Yaskawa INFORM job: TWIN_FRONT_WELD_90ST-2_5340.JBI

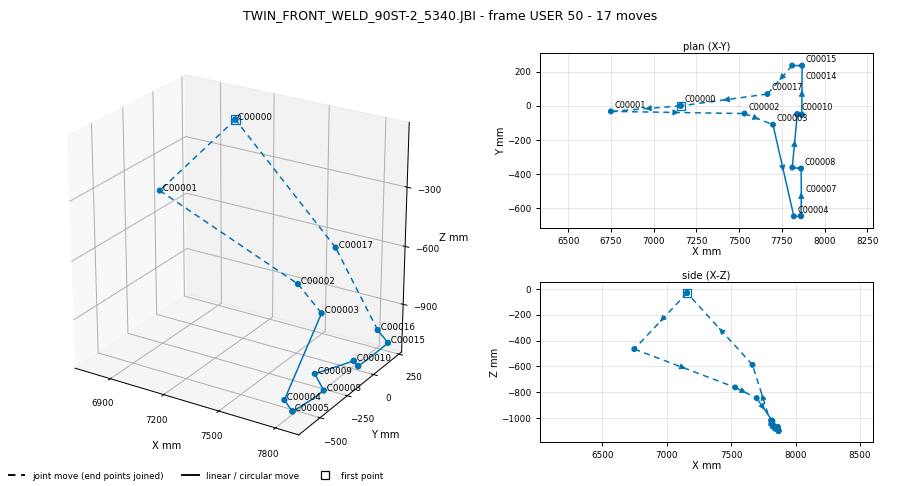
[picture p0: tool path of TWIN_FRONT_WELD_90ST-2_5340.JBI in frame USER 50, 17 of 19 moves have a stored position in this frame; points joined in program order, loops and branches not executed]
/JOB
//NAME TWIN_FRONT_WELD_90ST-2_5340
///FOLDERNAME 02-SKRZYNIE_JOBS
//POS
///NPOS 19,19,0,4,0,0
///USER 50
///TOOL 0
///POSTYPE USER
///RECTAN
///RCONF 0,0,1,0,0,0,0,0,0,0,0,0,0,0,0,0,0,0,0,0,0,0,0,0
C00000=7158.107,0.308,-30.113,-0.0036,-53.6521,0.0034
///RCONF 1,0,1,0,0,0,0,0,0,0,0,0,0,0,0,0,0,0,0,0,0,0,0,0
C00001=6749.261,-32.286,-465.417,15.1595,35.6819,-145.6807
///RCONF 1,0,0,0,0,0,0,0,0,0,0,0,0,0,0,0,0,0,0,0,0,0,0,0
C00002=7531.538,-44.927,-762.719,8.7291,34.6461,-164.2133
C00003=7698.169,-109.933,-845.445,15.9625,40.0165,-157.0814
///RCONF 0,0,0,0,0,0,0,0,0,0,0,0,0,0,0,0,0,0,0,0,0,0,0,0
C00004=7820.412,-646.733,-1023.988,41.9712,23.9862,-139.0909
C00005=7861.855,-645.939,-1070.027,41.9679,23.9849,-139.0942
C00006=7861.883,-644.400,-1070.166,41.9241,23.9457,-138.9976
C00007=7863.853,-523.749,-1081.452,38.5881,21.3794,-131.1067
C00008=7862.327,-366.605,-1089.610,38.1696,21.1192,-130.0311
C00009=7811.247,-360.951,-1020.499,38.1489,21.1058,-129.9915
C00010=7840.461,-48.547,-1081.078,15.4598,43.5968,-152.6291
C00011=7840.461,-48.547,-1081.078,15.4598,43.5968,-152.6291
C00012=7866.884,-53.201,-1100.385,16.0624,44.4125,-152.2042
C00013=7866.872,-51.635,-1100.322,16.0493,44.3951,-152.2149
C00014=7868.115,138.390,-1101.845,15.6338,43.8142,-152.4976
C00015=7868.719,235.750,-1099.768,15.4205,43.5150,-152.6513
C00016=7810.551,236.362,-1047.059,12.8910,39.7294,-154.3361
C00017=7665.720,69.333,-587.847,56.5185,9.2692,-73.1107
///RCONF 0,0,1,0,0,0,0,0,0,0,0,0,0,0,0,0,0,0,0,0,0,0,0,0
C00018=7158.107,0.308,-30.113,-0.0036,-53.6521,0.0034
///RCONF 0,0,0,0,0,0,0,0,0,0,0,0,0,0,0,0,0,0,0,0,0,0,0,0
BC00000=5343.689
BC00001=5343.689
BC00002=6178.800
BC00003=6495.017
BC00004=6688.143
BC00005=6688.143
BC00006=6688.143
BC00007=6688.143
BC00008=6688.143
BC00009=6688.143
BC00010=6686.021
BC00011=6686.021
BC00012=6686.021
BC00013=6686.021
BC00014=6686.021
BC00015=6686.021
BC00016=6686.021
BC00017=6015.470
BC00018=5343.689
///POSTYPE BASE
P00501=-2.026,0.009,3.534,0.0000,0.0000,0.0000
///RCONF 1,0,0,0,0,0,0,0,0,0,0,0,0,0,0,0,0,0,0,0,0,0,0,0
P00502=-2.023,0.001,1.732,0.0000,0.0000,0.0000
P00503=0.138,-0.044,1.539,0.0000,0.0000,0.0000
P00504=-0.309,-0.010,1.636,0.0000,0.0000,0.0000
//INST
///DATE 2024/10/29 10:05
///ATTR SC,RW,RJ
////FRAME USER 50
///GROUP1 RB1,BS1
NOP
MOVJ C00000 BC00000 VJ=50.00
MOVJ C00001 BC00001 VJ=50.00
MOVJ C00002 BC00002 VJ=50.00
MOVJ C00003 BC00003 VJ=50.00
'::::::::::::::::::::::::::::::::
'W56
'::::::::::::::::::::::::::::::::
MOVL C00004 BC00004 V=666.7
SFTON P0501
MACRO1 MJ#(0) ARGF14
MOVL C00005 BC00005 V=166.7 PL=0
ARCON
MOVC C00006 BC00006 V=9.5
MOVC C00007 BC00007 V=9.5
SFTOF
SFTON P0502
MOVC C00008 BC00008 V=9.5
ARCOF
MOVL C00009 BC00009 V=333.3
SFTOF
MOVL C00010 BC00010 V=333.3
'::::::::::::::::::::::::::::::::
'W21
'::::::::::::::::::::::::::::::::
MOVL C00011 BC00011 V=166.7
SFTON P0503
MACRO1 MJ#(0) ARGF14
MOVL C00012 BC00012 V=166.7 PL=0
ARCON
MOVC C00013 BC00013 V=9.5
SFTOF
SFTON P0504
MOVC C00014 BC00014 V=9.5
MOVC C00015 BC00015 V=9.5
ARCOF
MOVL C00016 BC00016 V=250.0
SFTOF
MOVJ C00017 BC00017 VJ=50.00
MOVJ C00018 BC00018 VJ=50.00
END
